    :  IF ((DI[26] OR DI[27]) AND F[324]),JMP LBL[53] ;
    :  IF ((!F[324] OR (TIMER[8]>=0)) AND ((F[523] AND !F[524] AND DI[2161]) OR (!F[523] AND F[524] AND !DI[2162])) AND DI[2167] AND F[576]),JMP LBL[54] ;
    :  IF ((!F[324] OR (TIMER[8]>=0)) AND ((F[523] AND !F[524] AND DI[2161]) OR (!F[523] AND F[524] AND !DI[2162])) AND !DI[2167] AND !F[576]),JMP LBL[54] ;
    :  R[42]=53    ;
    :   ;
    :  !**************************** ;
    :  !*        Schritt 54        * ;
    :  !*       MS1 Reinigung      * ;
    :  !* MS1 in Ruhest. schwenken * ;
    :  !**************************** ;
    :   ;
    :  LBL[54] ;
    :  R[41]=54    ;
    :  DO[2167]=(OFF) ;
    :  !Steuerluft EIN ;
    :  DO[2161]=(ON) ;
    :  !Schwenkeinheit 1 in Ruhestellung ;
    :  DO[2163]=(!DI[2163]) ;
    :  DO[2164]=(OFF) ;
    :  !FRG Bewegung EIN ;
    :  DO[2165]=(OFF) ;
    :  DO[2166]=(!DI[2163]) ;
    :  DO[18181]=(ON) ;
    :  WAIT (!DI[2164] AND DI[2163])    ;
    :  DO[18181]=(OFF) ;
    :  !RSK Fehlerausgabe Schwenkeinheit ;
    :  F[323]=((!DI[2163] AND (TIMER[8]>=0)) OR F[323]) ;
    :  !RSK Sammelstoerung ;
    :  F[329]=(F[323]) ;
    :  DO[2163]=(OFF) ;
    :  DO[2164]=(OFF) ;
    :  !FRG Bewegung AUS ;
    :  DO[2166]=(OFF) ;
    :  IF (F[323] AND (DI[26] OR DI[27])),JMP LBL[47] ;
    :  DO[18181]=(ON) ;
    :  WAIT (!F[323] AND DI[2165])    ;
    :  DO[18181]=(OFF) ;
    :  F[323]=(OFF) ;
    :  F[329]=(OFF) ;
    :  !FRG in Endlage halten ein ;
    :  DO[2165]=(ON) ;
    :  DO[18181]=(ON) ;
    :  WAIT   2.00(sec) ;
    :  WAIT (!DI[2165])    ;
    :  DO[18181]=(OFF) ;
    :  !Steuerluft AUS ;
    :  DO[2161]=(OFF) ;
    :  !FRG in Endlage halten AUS ;
    :  DO[2165]=(OFF) ;
    :  !MS1 Zaehler ruecksetzen ;
    :  R[21]=0    ;
    :  !MS1 FRG Reinigung ;
    :  F[603]=(OFF) ;
    :  !MS1 Reinigung FK ;
    :  F[605]=(ON) ;
    :  R[42]=54    ;
    :  JMP LBL[1] ;
    :   ;
    :  !************************** ;
    :  !*       Schritt 55       * ;
    :  !*      STAT EZ1/SP1      * ;
    :  !* 2.Setzhub nach Fraesen * ;
    :  !************************** ;
    :   ;
    :  LBL[55] ;
    :  R[41]=55    ;
    :  !RSK gestartet ;
    :  F[321]=(OFF) ;
    :  !EZ1/SK1 Prog. ;
    :  IF (F[78]),GO[1]=(61) ;
    :  IF (F[78]),GO[3]=(61) ;
    :  WAIT    .10(sec) ;
    :  !EZ1/SP1 schliessen ;
    :  DO[717]=(OFF) ;
    :  DO[718]=(ON) ;
    :  TIMER[9]=((-8)) ;
    :  !EZ1/SP1 Kraft erreicht ;
    :  WAIT ((DI[718] AND !DI[717]) OR (TIMER[9]>=0))    ;
    :  DO[18181]=((TIMER[9]>=0)) ;
    :  WAIT (DI[718] AND !DI[717])    ;
    :  DO[18181]=(OFF) ;
    :  WAIT   1.00(sec) ;
    :  !EZ1/SP1 oeffnen ;
    :  DO[718]=(OFF) ;
    :  DO[717]=(!DI[717]) ;
    :  TIMER[9]=((-8)) ;
    :  WAIT (DI[717] OR (TIMER[9]>=0))    ;
    :  DO[18181]=((TIMER[9]>=0)) ;
    :  WAIT (DI[717])    ;
    :  DO[18181]=(OFF) ;
    :  DO[717]=(OFF) ;
    :  R[42]=55    ;
    :  JMP LBL[16] ;
    :   ;
    :  !************************** ;
    :  !*       Schritt 56       * ;
    :  !*      STAT EZ2/SP2      * ;
    :  !* 2.Setzhub nach Fraesen * ;
    :  !************************** ;
    :   ;
    :  LBL[56] ;
    :  R[41]=56    ;
    :  !RSK gestartet ;
    :  F[321]=(OFF) ;
    :  !EZ2/SK2 Prog. ;
    :  IF (F[285] AND F[138]),GO[3]=(65) ;
    :  IF (!F[285] AND F[138]),GO[4]=(61) ;
    :  IF (!F[285] AND F[138]),GO[6]=(61) ;
    :  WAIT    .10(sec) ;
    :  !EZ2/SP2 schliessen ;
    :  DO[877]=(OFF) ;
    :  DO[878]=(ON) ;
    :  TIMER[9]=((-8)) ;
    :  !EZ2/SP2 Kraft erreicht ;
    :  WAIT ((DI[878] AND !DI[877]) OR (TIMER[9]>=0))    ;
    :  DO[18181]=((TIMER[9]>=0)) ;
    :  WAIT (DI[878] AND !DI[877])    ;
    :  DO[18181]=(OFF) ;
    :  WAIT   1.00(sec) ;
    :  !EZ2/SP2 oeffnen ;
    :  DO[878]=(OFF) ;
    :  DO[877]=(!DI[877]) ;
    :  TIMER[9]=((-8)) ;
    :  WAIT (DI[877] OR (TIMER[9]>=0))    ;
    :  DO[18181]=((TIMER[9]>=0)) ;
    :  WAIT (DI[877])    ;
    :  DO[18181]=(OFF) ;
    :  DO[877]=(OFF) ;
    :  R[42]=56    ;
    :  JMP LBL[25] ;
    :   ;
    :  !************************** ;
    :  !*       Schritt 57       * ;
    :  !*      STAT EZ3/SP3      * ;
    :  !* 2.Setzhub nach Fraesen * ;
    :  !************************** ;
    :   ;
    :  LBL[57] ;
    :  R[41]=57    ;
    :  !RSK gestartet ;
    :  F[321]=(OFF) ;
    :  !EZ1/SK1 Prog. ;
    :  IF (F[174]),GO[7]=(61) ;
    :  IF (F[174]),GO[9]=(61) ;
    :  WAIT    .10(sec) ;
    :  !EZ3/SP3 schliessen ;
    :  DO[1037]=(OFF) ;
    :  DO[1038]=(ON) ;
    :  TIMER[9]=((-8)) ;
    :  !EZ3/SP3 Kraft erreicht ;
    :  WAIT ((DI[1038] AND !DI[1037]) OR (TIMER[9]>=0))    ;
    :  DO[18181]=((TIMER[9]>=0)) ;
    :  WAIT (DI[1038] AND !DI[1037])    ;
    :  DO[18181]=(OFF) ;
    :  WAIT   1.00(sec) ;
    :  !EZ3/SP3 oeffnen ;
    :  DO[1038]=(OFF) ;
    :  DO[1037]=(!DI[1037]) ;
    :  TIMER[9]=((-8)) ;
    :  WAIT (DI[1037] OR (TIMER[9]>=0))    ;
    :  DO[18181]=((TIMER[9]>=0)) ;
    :  WAIT (DI[1037])    ;
    :  DO[18181]=(OFF) ;
    :  DO[1037]=(OFF) ;
    :  R[42]=57    ;
    :  JMP LBL[34] ;
    :   ;
    :  !*************************** ;
    :  !*************************** ;
    :  !* Fraesen Rob EZ1 SZ1-SZ4 * ;
    :  !*          an KF2         * ;
    :  !*************************** ;
    :  !*************************** ;
    :   ;
    :   ;
    :  !**************************** ;
    :  !*        Schritt 58        * ;
    :  !* Rob EZ1 SZ1-SZ4 Auswert. * ;
    :  !**************************** ;
    :   ;
    :  LBL[58] ;
    :  R[41]=58    ;
    :  !RSK gestartet ;
    :  F[321]=(OFF) ;
    :  GO[1]=(31) ;
    :  IF (F[64]),GO[3]=(31) ;
    :  IF (F[65]),GO[3]=(32) ;
    :  IF (F[66]),GO[3]=(33) ;
    :  IF (F[67]),GO[3]=(34) ;
    :  WAIT    .10(sec) ;
    :  DO[116]=(ON) ;
    :  DO[130]=(ON) ;
    :  DO[718]=(OFF) ;
    :  DO[717]=(!DI[717]) ;
    :  DO[18181]=(ON) ;
    :  WAIT (DI[717])    ;
    :  DO[18181]=(OFF) ;
    :  DO[717]=(OFF) ;
    :  !Anwahl Startfraesen ;
    :  IF (F[90] AND F[78] AND !F[79]),R[41]=59 ;
    :  !Anwahl Normalfraesen ;
    :  IF (F[90] AND !F[78] AND F[79]),R[41]=61 ;
    :  R[42]=58    ;
    :  JMP LBL[R[41]] ;
    :   ;
    :  !***************************** ;
    :  !*         Schritt 59        * ;
    :  !* Rob EZ1 SZ1-SZ4 SF Teil 1 * ;
    :  !***************************** ;
    :   ;
    :  LBL[59] ;
    :  R[41]=59    ;
    :  !RSK gestartet ;
    :  F[321]=(OFF) ;
    :  F[329]=(OFF) ;
    :  F[325]=(OFF) ;
    :  DO[718]=(OFF) ;
    :  DO[717]=(!DI[717]) ;
    :  DO[18181]=(ON) ;
    :  WAIT (DI[717])    ;
    :  DO[18181]=(OFF) ;
    :  DO[994]=(ON) ;
    :  DO[717]=(OFF) ;
    :  !Warte Fraeser laeuft ;
    :  TIMER[7]=((-3)) ;
    :  WAIT (!DI[994] OR (TIMER[7]>=0))    ;
    :  WAIT (DI[994] OR (TIMER[7]>=0))    ;
    :  F[322]=((TIMER[7]>=0)) ;
    :  DO[18181]=(ON) ;
    :  WAIT (!DI[994])    ;
    :  WAIT (DI[994])    ;
    :  DO[18181]=(OFF) ;
    :  F[322]=(OFF) ;
    :  !EZ1/SP1 schliessen ;
    :  DO[718]=(ON) ;
    :  TIMER[9]=((-4)) ;
    :  !EZ1/SP1 Kraft erreicht ;
    :  WAIT ((DI[718] AND !DI[772] AND !DI[780] AND !DI[774] AND !DI[775]) OR (TIMER[9]>=0))    ;
    :  DO[18181]=(ON) ;
    :  DO[718]=((TIMER[9]<0)) ;
    :  DO[994]=((TIMER[9]<0)) ;
    :  WAIT ((DI[718] AND !DI[772] AND !DI[780] AND !DI[774] AND !DI[775]) OR DI[26] OR DI[27])    ;
    :  F[325]=(DI[26] OR DI[27]) ;
    :  DO[18181]=(OFF) ;
    :  !EZ1/SP1 Fehler Kraftaufbau ;
    :  IF (F[325]),JMP LBL[5906] ;
    :  TIMER[9]=((-5)) ;
    :  LBL[5900] ;
    :  WAIT (!DI[994] OR F[325] OR (TIMER[9]>=0))    ;
    :  WAIT (DI[994] OR F[325] OR (TIMER[9]>=0))    ;
    :  R[1]=(R[1]+1) ;
    :  F[329]=((TIMER[9]>=0)) ;
    :  !Fraeszeit ueberschritten ;
    :  IF (F[329]),JMP LBL[5906] ;
    :  IF (F[64]),JMP LBL[5902] ;
    :  IF (F[65]),JMP LBL[5903] ;
    :  IF (F[66]),JMP LBL[5904] ;
    :  IF (F[67]),JMP LBL[5905] ;
    :  !Umdrehungen Vergl.SZ1 ;
    :  LBL[5902] ;
    :  !Umdrehungen Vergleichen ;
    :  IF (R[1]<R[2]),JMP LBL[5900] ;
    :  JMP LBL[5901] ;
    :  !Umdrehungen Vergl.SZ2 ;
    :  LBL[5903] ;
    :  !Umdrehungen Vergleichen ;
    :  IF (R[1]<R[8]),JMP LBL[5900] ;
    :  JMP LBL[5901] ;
    :  !Umdrehungen Vergl.SZ3 ;
    :  LBL[5904] ;
    :  !Umdrehungen Vergleichen ;
    :  IF (R[1]<R[11]),JMP LBL[5900] ;
    :  JMP LBL[5901] ;
    :  !Umdrehungen Vergl.SZ4 ;
    :  LBL[5905] ;
    :  !Umdrehungen Vergleichen ;
    :  IF (R[1]<R[14]),JMP LBL[5900] ;
    :  JMP LBL[5901] ;
    :  LBL[5901] ;
    :  IF (F[64]),F[94]=(ON) ;
    :  IF (F[65]),F[100]=(ON) ;
    :  IF (F[66]),F[106]=(ON) ;
    :  IF (F[67]),F[112]=(ON) ;
    :  LBL[5906] ;
    :  DO[994]=((TIMER[9]<0)) ;
    :  !Fraeser ausblasen EIN ;
    :  DO[995]=((TIMER[9]<0)) ;
    :  DO[718]=(OFF) ;
    :  !EZ1/SP1 oeffnen ;
    :  DO[717]=(!DI[717]) ;
    :  DO[18181]=(F[329]) ;
    :  WAIT (!F[329] OR DI[26] OR DI[27])    ;
    :  DO[18181]=(OFF) ;
    :  DO[18181]=(ON) ;
    :  WAIT (DI[717])    ;
    :  DO[18181]=(OFF) ;
    :  DO[717]=(OFF) ;
    :  !Umdrehungen ruecksetzen ;
    :  R[1]=0    ;
    :  R[42]=59    ;
    :  IF (F[329] OR F[325]),JMP LBL[59] ;
    :  JMP LBL[60] ;
    :   ;
    :  !***************************** ;
    :  !*         Schritt 60        * ;
    :  !* Rob EZ1 SZ1-SZ4 SF Teil 2 * ;
    :  !***************************** ;
    :   ;
    :  LBL[60] ;
    :  R[41]=60    ;
    :  !RSK gestartet ;
    :  F[321]=(OFF) ;
    :  F[329]=(OFF) ;
    :  F[325]=(OFF) ;
    :  DO[718]=(OFF) ;
    :  DO[717]=(!DI[717]) ;
    :  DO[18181]=(ON) ;
    :  WAIT (DI[717])    ;
    :  DO[18181]=(OFF) ;
    :  DO[994]=(ON) ;
    :  DO[717]=(OFF) ;
    :  !EZ1/SP1 schliessen ;
    :  DO[718]=(ON) ;
    :  !Fraeser ausblasen AUS ;
    :  DO[995]=(OFF) ;
    :  TIMER[9]=((-4)) ;
    :  !EZ1/SP1 Kraft erreicht ;
    :  WAIT ((DI[718] AND !DI[772] AND !DI[780] AND !DI[774] AND !DI[775]) OR (TIMER[9]>=0))    ;
    :  DO[18181]=(ON) ;
    :  DO[718]=((TIMER[9]<0)) ;
    :  DO[994]=((TIMER[9]<0)) ;
    :  WAIT ((DI[718] AND !DI[772] AND !DI[780] AND !DI[774] AND !DI[775]) OR DI[26] OR DI[27])    ;
    :  F[325]=(DI[26] OR DI[27]) ;
    :  DO[18181]=(OFF) ;
    :  !EZ1/SP1 Fehler Kraftaufbau ;
    :  IF (F[325]),JMP LBL[60] ;
    :  TIMER[9]=((-5)) ;
    :  LBL[6000] ;
    :  WAIT (!DI[994] OR F[325] OR (TIMER[9]>=0))    ;
    :  WAIT (DI[994] OR F[325] OR (TIMER[9]>=0))    ;
    :  R[1]=(R[1]+1) ;
    :  F[329]=((TIMER[9]>=0)) ;
    :  !Fraeszeit ueberschritten ;
    :  IF (F[329]),JMP LBL[6006] ;
    :  IF (F[64]),JMP LBL[6002] ;
    :  IF (F[65]),JMP LBL[6003] ;
    :  IF (F[66]),JMP LBL[6004] ;
    :  IF (F[67]),JMP LBL[6005] ;
    :  !Umdrehungen Vergl.SZ1 ;
    :  LBL[6002] ;
    :  !Umdrehungen Vergleichen ;
    :  IF (R[1]<R[3]),JMP LBL[6000] ;
    :  JMP LBL[6001] ;
    :  !Umdrehungen Vergl.SZ2 ;
    :  LBL[6003] ;
    :  !Umdrehungen Vergleichen ;
    :  IF (R[1]<R[9]),JMP LBL[6000] ;
    :  JMP LBL[6001] ;
    :  !Umdrehungen Vergl.SZ3 ;
    :  LBL[6004] ;
    :  !Umdrehungen Vergleichen ;
    :  IF (R[1]<R[12]),JMP LBL[6000] ;
    :  JMP LBL[6001] ;
    :  !Umdrehungen Vergl.SZ4 ;
    :  LBL[6005] ;
    :  !Umdrehungen Vergleichen ;
    :  IF (R[1]<R[15]),JMP LBL[6000] ;
    :  JMP LBL[6001] ;
    :  LBL[6001] ;
    :  IF (F[64]),F[96]=(ON) ;
    :  IF (F[65]),F[102]=(ON) ;
    :  IF (F[66]),F[108]=(ON) ;
    :  IF (F[67]),F[114]=(ON) ;
    :  LBL[6006] ;
    :  DO[994]=((TIMER[9]<0)) ;
    :  !Fraeser ausblasen EIN ;
    :  IF ((TIMER[9]<0)),DO[995]=PULSE,3.0sec ;
    :  DO[718]=(OFF) ;
    :  !EZ1/SP1 oeffnen ;
    :  DO[717]=(!DI[717]) ;
    :  DO[18181]=(F[329]) ;
    :  WAIT (!F[329] OR DI[26] OR DI[27])    ;
    :  DO[18181]=(OFF) ;
    :  DO[18181]=(ON) ;
    :  WAIT (DI[717])    ;
    :  DO[18181]=(OFF) ;
    :  DO[717]=(OFF) ;
    :  !Umdrehungen ruecksetzen ;
    :  R[1]=0    ;
    :  R[42]=60    ;
    :  IF (F[329] OR F[325]),JMP LBL[60] ;
    :  JMP LBL[62] ;
    :   ;
    :  !********************** ;
    :  !*     Schritt 61      * ;
    :  !* Rob EZ1 SZ1-SZ4 NF * ;
    :  !********************** ;
    :   ;
    :  LBL[61] ;
    :  R[41]=61    ;
    :  !RSK gestartet ;
    :  F[321]=(OFF) ;
    :  F[329]=(OFF) ;
    :  F[325]=(OFF) ;
    :  DO[718]=(OFF) ;
    :  DO[717]=(!DI[717]) ;
    :  DO[18181]=(ON) ;
    :  WAIT (DI[717])    ;
    :  DO[18181]=(OFF) ;
    :  DO[994]=(ON) ;
    :  DO[717]=(OFF) ;
    :  !Warte Fraeser laeuft ;
    :  TIMER[7]=((-3)) ;
    :  WAIT (!DI[994] OR (TIMER[7]>=0))    ;
    :  WAIT (DI[994] OR (TIMER[7]>=0))    ;
    :  F[322]=((TIMER[7]>=0)) ;
    :  DO[18181]=(ON) ;
    :  WAIT (!DI[994])    ;
    :  WAIT (DI[994])    ;
    :  DO[18181]=(OFF) ;
    :  F[322]=(OFF) ;
    :  !EZ1/SP1 schliessen ;
    :  DO[718]=(ON) ;
    :  TIMER[9]=((-4)) ;
    :  !EZ1/SP1 Kraft erreicht ;
    :  WAIT ((DI[718] AND !DI[772] AND !DI[780] AND !DI[774] AND !DI[775]) OR (TIMER[9]>=0))    ;
    :  DO[18181]=(ON) ;
    :  DO[718]=((TIMER[9]<0)) ;
    :  DO[994]=((TIMER[9]<0)) ;
    :  WAIT ((DI[718] AND !DI[772] AND !DI[780] AND !DI[774] AND !DI[775]) OR DI[26] OR DI[27])    ;
    :  F[325]=(DI[26] OR DI[27]) ;
    :  DO[18181]=(OFF) ;
    :  !EZ1/SP1 Fehler Kraftaufbau ;
    :  IF (F[325]),JMP LBL[61] ;
    :  TIMER[9]=((-5)) ;
    :  LBL[6100] ;
    :  WAIT (!DI[994] OR F[325] OR (TIMER[9]>=0))    ;
    :  WAIT (DI[994] OR F[325] OR (TIMER[9]>=0))    ;
    :  R[1]=(R[1]+1) ;
    :  F[329]=((TIMER[9]>=0)) ;
    :  !Fraeszeit ueberschritten ;
    :  IF (F[329]),JMP LBL[6106] ;
    :  IF (F[64]),JMP LBL[6102] ;
    :  IF (F[65]),JMP LBL[6103] ;
    :  IF (F[66]),JMP LBL[6104] ;
    :  IF (F[67]),JMP LBL[6105] ;
    :  !Umdrehungen Vergl.SZ1 ;
    :  LBL[6102] ;
    :  !Umdrehungen Vergleichen ;
    :  IF (R[1]<R[4]),JMP LBL[6100] ;
    :  JMP LBL[6101] ;
    :  !Umdrehungen Vergl.SZ2 ;
    :  LBL[6103] ;
    :  !Umdrehungen Vergleichen ;
    :  IF (R[1]<R[10]),JMP LBL[6100] ;
    :  !Umdrehungen Vergl.SZ3 ;
    :  LBL[6104] ;
    :  !Umdrehungen Vergleichen ;
    :  IF (R[1]<R[13]),JMP LBL[6100] ;
    :  JMP LBL[6101] ;
    :  !Umdrehungen Vergl.SZ4 ;
    :  LBL[6105] ;
    :  !Umdrehungen Vergleichen ;
    :  IF (R[1]<R[16]),JMP LBL[6100] ;
    :  LBL[6101] ;
    :  !EZ1/SP1 2 Huebe bei NF ;
    :  IF (!F[130]),JMP LBL[6106] ;
    :  IF (F[98]),F[96]=(ON) ;
    :  IF (F[104]),F[96]=(ON) ;
    :  IF (F[110]),F[96]=(ON) ;
    :  IF (F[116]),F[96]=(ON) ;
    :  IF (F[64]),F[98]=(ON) ;
    :  IF (F[65]),F[104]=(ON) ;
    :  IF (F[66]),F[110]=(ON) ;
    :  IF (F[67]),F[116]=(ON) ;
    :  LBL[6106] ;
    :  DO[994]=((TIMER[9]<0)) ;
    :  !Fraeser ausblasen EIN ;
    :  IF ((TIMER[9]<0)),DO[995]=PULSE,3.0sec ;
    :  DO[718]=(OFF) ;
    :  !EZ1/SP1 oeffnen ;
    :  DO[717]=(!DI[717]) ;
    :  DO[18181]=(F[329]) ;
    :  WAIT (!F[329] OR DI[26] OR DI[27])    ;
    :  DO[18181]=(OFF) ;
    :  DO[18181]=(ON) ;
    :  WAIT (DI[717])    ;
    :  DO[18181]=(OFF) ;
    :  DO[717]=(OFF) ;
    :  !Umdrehungen ruecksetzen ;
    :  R[1]=0    ;
    :  R[42]=61    ;
    :  IF (F[329] OR (!F[96] AND F[130])),JMP LBL[61] ;
    :  IF (F[64]),F[98]=(ON) ;
    :  IF (F[65]),F[104]=(ON) ;
    :  IF (F[66]),F[110]=(ON) ;
    :  IF (F[67]),F[116]=(ON) ;
    :  JMP LBL[62] ;
    :   ;
    :  !******************************* ;
    :  !*         Schritt 62          * ;
    :  !* Rob EZ1 SZ1-SZ4 i.O./n.i.O. * ;
    :  !******************************* ;
    :   ;
    :  LBL[62] ;
    :  R[41]=62    ;
    :  !Fraesueberwachung starten ;
    :  IF (F[64]),JMP LBL[6201] ;
    :  IF (F[65]),JMP LBL[6202] ;
    :  IF (F[66]),JMP LBL[6203] ;
    :  IF (F[67]),JMP LBL[6204] ;
    :  LBL[6201] ;
    :  TIMER[7]=((-3)) ;
    :  WAIT (F[64] AND ((F[79] AND F[98]) OR (F[78] AND F[94] AND F[96])) OR (TIMER[7]>=0))    ;
    :  F[329]=((TIMER[7]>=0)) ;
    :  DO[18181]=(ON) ;
    :  WAIT (F[64] AND ((F[79] AND F[98]) OR (F[78] AND F[94] AND F[96])))    ;
    :  DO[18181]=(OFF) ;
    :  JMP LBL[6200] ;
    :  LBL[6202] ;
    :  TIMER[7]=((-3)) ;
    :  WAIT (F[65] AND ((F[79] AND F[104]) OR (F[78] AND F[100] AND F[102])) OR (TIMER[7]>=0))    ;
    :  F[329]=((TIMER[7]>=0)) ;
    :  DO[18181]=(ON) ;
    :  WAIT (F[65] AND ((F[79] AND F[104]) OR (F[78] AND F[100] AND F[102])))    ;
    :  DO[18181]=(OFF) ;
    :  JMP LBL[6200] ;
    :  LBL[6203] ;
    :  TIMER[7]=((-3)) ;
    :  WAIT (F[66] AND ((F[79] AND F[110]) OR (F[78] AND F[106] AND F[108])) OR (TIMER[7]>=0))    ;
    :  F[329]=((TIMER[7]>=0)) ;
    :  DO[18181]=(ON) ;
    :  WAIT (F[66] AND ((F[79] AND F[110]) OR (F[78] AND F[106] AND F[108])))    ;
    :  DO[18181]=(OFF) ;
    :  JMP LBL[6200] ;
    :  LBL[6204] ;
    :  TIMER[7]=((-3)) ;
    :  WAIT (F[67] AND ((F[79] AND F[116]) OR (F[78] AND F[112] AND F[114])) OR (TIMER[7]>=0))    ;
    :  F[329]=((TIMER[7]>=0)) ;
    :  DO[18181]=(ON) ;
    :  WAIT (F[67] AND ((F[79] AND F[116]) OR (F[78] AND F[112] AND F[114])))    ;
    :  DO[18181]=(OFF) ;
    :  JMP LBL[6200] ;
    :  LBL[6200] ;
    :  R[41]=63    ;
    :  !KF1 U-Merker ruecksetzen ;
    :  F[94]=(OFF) ;
    :  F[96]=(OFF) ;
    :  F[98]=(OFF) ;
    :  F[100]=(OFF) ;
    :  F[102]=(OFF) ;
    :  F[104]=(OFF) ;
    :  F[106]=(OFF) ;
    :  F[108]=(OFF) ;
    :  F[110]=(OFF) ;
    :  F[112]=(OFF) ;
    :  F[114]=(OFF) ;
    :  F[116]=(OFF) ;
    :  R[42]=62    ;
    :  JMP LBL[R[41]] ;
    :   ;
    :  !***************************** ;
    :  !*        Schritt 63         * ;
    :  !* Rob EZ1 SZ1-SZ4 Quitt SK1 * ;
    :  !***************************** ;
    :   ;
    :  LBL[63] ;
    :  R[41]=63    ;
    :  !RSK gestartet ;
    :  F[321]=(OFF) ;
    :  IF (F[64]),GO[3]=1 ;
    :  IF (F[65]),GO[3]=2 ;
    :  IF (F[66]),GO[3]=3 ;
    :  IF (F[67]),GO[3]=4 ;
    :  WAIT    .10(sec) ;
    :  DO[786]=(ON) ;
    :  DO[116]=(OFF) ;
    :  DO[130]=(OFF) ;
    :  DO[18181]=(ON) ;
    :  WAIT (!DI[786] AND DI[787] AND !DI[788])    ;
    :  !FK Fraesen ;
    :  F[91]=(!F[329]) ;
    :  DO[18181]=(OFF) ;
    :  DO[786]=(OFF) ;
    :  R[42]=63    ;
    :  JMP LBL[1] ;
    :   ;
    :  !*************************** ;
    :  !*************************** ;
    :  !* Fraesen Rob EZ1 SZ1-SZ4 * ;
    :  !*          an KF3         * ;
    :  !*************************** ;
    :  !*************************** ;
    :   ;
    :   ;
    :  !**************************** ;
    :  !*        Schritt 64        * ;
    :  !* Rob EZ1 SZ1-SZ4 Auswert. * ;
    :  !**************************** ;
    :   ;
    :  LBL[64] ;
    :  R[41]=64    ;
    :  !RSK gestartet ;
    :  F[321]=(OFF) ;
    :  GO[1]=(31) ;
    :  IF (F[64]),GO[3]=(31) ;
    :  IF (F[65]),GO[3]=(32) ;
    :  IF (F[66]),GO[3]=(33) ;
    :  IF (F[67]),GO[3]=(34) ;
    :  WAIT    .10(sec) ;
    :  DO[116]=(ON) ;
    :  DO[130]=(ON) ;
    :  DO[718]=(OFF) ;
    :  DO[717]=(!DI[717]) ;
    :  DO[18181]=(ON) ;
    :  WAIT (DI[717])    ;
    :  DO[18181]=(OFF) ;
    :  DO[717]=(OFF) ;
    :  !Anwahl Startfraesen ;
    :  IF (F[90] AND F[78] AND !F[79]),R[41]=65 ;
    :  !Anwahl Normalfraesen ;
    :  IF (F[90] AND !F[78] AND F[79]),R[41]=67 ;
    :  R[42]=64    ;
    :  JMP LBL[R[41]] ;
    :   ;
    :  !***************************** ;
    :  !*         Schritt 65        * ;
    :  !* Rob EZ1 SZ1-SZ4 SF Teil 1 * ;
    :  !***************************** ;
    :   ;
    :  LBL[65] ;
    :  R[41]=65    ;
    :  !RSK gestartet ;
    :  F[321]=(OFF) ;
    :  F[329]=(OFF) ;
    :  F[325]=(OFF) ;
    :  DO[718]=(OFF) ;
    :  DO[717]=(!DI[717]) ;
    :  DO[18181]=(ON) ;
    :  WAIT (DI[717])    ;
    :  DO[18181]=(OFF) ;
    :  DO[1154]=(ON) ;
    :  DO[717]=(OFF) ;
    :  !Warte Fraeser laeuft ;
    :  TIMER[7]=((-3)) ;
    :  WAIT (!DI[1154] OR (TIMER[7]>=0))    ;
    :  WAIT (DI[1154] OR (TIMER[7]>=0))    ;
    :  F[322]=((TIMER[7]>=0)) ;
    :  DO[18181]=(ON) ;
    :  WAIT (!DI[1154])    ;
    :  WAIT (DI[1154])    ;
    :  DO[18181]=(OFF) ;
    :  F[322]=(OFF) ;
    :  !EZ1/SP1 schliessen ;
    :  DO[718]=(ON) ;
    :  TIMER[9]=((-4)) ;
    :  !EZ1/SP1 Kraft erreicht ;
    :  WAIT ((DI[718] AND !DI[772] AND !DI[780] AND !DI[774] AND !DI[775]) OR (TIMER[9]>=0))    ;
    :  DO[18181]=(ON) ;
    :  DO[718]=((TIMER[9]<0)) ;
    :  DO[1154]=((TIMER[9]<0)) ;
    :  WAIT ((DI[718] AND !DI[772] AND !DI[780] AND !DI[774] AND !DI[775]) OR DI[26] OR DI[27])    ;
    :  F[325]=(DI[26] OR DI[27]) ;
    :  DO[18181]=(OFF) ;
    :  !EZ1/SP1 Fehler Kraftaufbau ;
    :  IF (F[325]),JMP LBL[6506] ;
    :  TIMER[9]=((-5)) ;
    :  LBL[6500] ;
    :  WAIT (!DI[1154] OR F[325] OR (TIMER[9]>=0))    ;
    :  WAIT (DI[1154] OR F[325] OR (TIMER[9]>=0))    ;
    :  R[1]=(R[1]+1) ;
    :  F[329]=((TIMER[9]>=0)) ;
    :  !Fraeszeit ueberschritten ;
    :  IF (F[329]),JMP LBL[6506] ;
    :  IF (F[64]),JMP LBL[6502] ;
    :  IF (F[65]),JMP LBL[6503] ;
    :  IF (F[66]),JMP LBL[6504] ;
    :  IF (F[67]),JMP LBL[6505] ;
    :  !Umdrehungen Vergl.SZ1 ;
    :  LBL[6502] ;
    :  !Umdrehungen Vergleichen ;
    :  IF (R[1]<R[2]),JMP LBL[6500] ;
    :  JMP LBL[6501] ;
    :  !Umdrehungen Vergl.SZ2 ;
    :  LBL[6503] ;
    :  !Umdrehungen Vergleichen ;
    :  IF (R[1]<R[8]),JMP LBL[6500] ;
    :  JMP LBL[6501] ;
    :  !Umdrehungen Vergl.SZ3 ;
    :  LBL[6504] ;
    :  !Umdrehungen Vergleichen ;
    :  IF (R[1]<R[11]),JMP LBL[6500] ;
    :  JMP LBL[6501] ;
    :  !Umdrehungen Vergl.SZ4 ;
    :  LBL[6505] ;
    :  !Umdrehungen Vergleichen ;
    :  IF (R[1]<R[14]),JMP LBL[6500] ;
    :  JMP LBL[6501] ;
    :  LBL[6501] ;
    :  IF (F[64]),F[94]=(ON) ;
    :  IF (F[65]),F[100]=(ON) ;
    :  IF (F[66]),F[106]=(ON) ;
    :  IF (F[67]),F[112]=(ON) ;
    :  LBL[6506] ;
    :  DO[1154]=((TIMER[9]<0)) ;
    :  !Fraeser ausblasen EIN ;
    :  DO[1155]=((TIMER[9]<0)) ;
    :  DO[718]=(OFF) ;
    :  !EZ1/SP1 oeffnen ;
    :  DO[717]=(!DI[717]) ;
    :  DO[18181]=(F[329]) ;
    :  WAIT (!F[329] OR DI[26] OR DI[27])    ;
    :  DO[18181]=(OFF) ;
    :  DO[18181]=(ON) ;
    :  WAIT (DI[717])    ;
    :  DO[18181]=(OFF) ;
    :  DO[717]=(OFF) ;
    :  !Umdrehungen ruecksetzen ;
    :  R[1]=0    ;
    :  R[42]=65    ;
    :  IF (F[329] OR F[325]),JMP LBL[65] ;
    :  JMP LBL[66] ;
    :   ;
    :  !***************************** ;
    :  !*         Schritt 66        * ;
    :  !* Rob EZ1 SZ1-SZ4 SF Teil 2 * ;
    :  !***************************** ;
    :   ;
    :  LBL[66] ;
    :  R[41]=66    ;
    :  !RSK gestartet ;
    :  F[321]=(OFF) ;
    :  F[329]=(OFF) ;
    :  F[325]=(OFF) ;
    :  DO[718]=(OFF) ;
    :  DO[717]=(!DI[717]) ;
    :  DO[18181]=(ON) ;
    :  WAIT (DI[717])    ;
    :  DO[18181]=(OFF) ;
    :  DO[1154]=(ON) ;
    :  DO[717]=(OFF) ;
    :  !EZ1/SP1 schliessen ;
    :  DO[718]=(ON) ;
    :  !Fraeser ausblasen AUS ;
    :  DO[1155]=(OFF) ;
    :  TIMER[9]=((-4)) ;
    :  !EZ1/SP1 Kraft erreicht ;
    :  WAIT ((DI[718] AND !DI[772] AND !DI[780] AND !DI[774] AND !DI[775]) OR (TIMER[9]>=0))    ;
    :  DO[18181]=(ON) ;
    :  DO[718]=((TIMER[9]<0)) ;
    :  DO[1154]=((TIMER[9]<0)) ;
    :  WAIT ((DI[718] AND !DI[772] AND !DI[780] AND !DI[774] AND !DI[775]) OR DI[26] OR DI[27])    ;
    :  F[325]=(DI[26] OR DI[27]) ;
    :  DO[18181]=(OFF) ;
    :  !EZ1/SP1 Fehler Kraftaufbau ;
    :  IF (F[325]),JMP LBL[66] ;
    :  TIMER[9]=((-5)) ;
    :  LBL[6600] ;
    :  WAIT (!DI[1154] OR F[325] OR (TIMER[9]>=0))    ;
    :  WAIT (DI[1154] OR F[325] OR (TIMER[9]>=0))    ;
    :  R[1]=(R[1]+1) ;
    :  F[329]=((TIMER[9]>=0)) ;
    :  !Fraeszeit ueberschritten ;
    :  IF (F[329]),JMP LBL[6606] ;
    :  IF (F[64]),JMP LBL[6602] ;
    :  IF (F[65]),JMP LBL[6603] ;
    :  IF (F[66]),JMP LBL[6604] ;
    :  IF (F[67]),JMP LBL[6605] ;
    :  !Umdrehungen Vergl.SZ1 ;
    :  LBL[6602] ;
    :  !Umdrehungen Vergleichen ;
    :  IF (R[1]<R[3]),JMP LBL[6600] ;
    :  JMP LBL[6601] ;
    :  !Umdrehungen Vergl.SZ2 ;
    :  LBL[6603] ;
    :  !Umdrehungen Vergleichen ;
    :  IF (R[1]<R[9]),JMP LBL[6600] ;
    :  JMP LBL[6601] ;
    :  !Umdrehungen Vergl.SZ3 ;
    :  LBL[6604] ;
    :  !Umdrehungen Vergleichen ;
    :  IF (R[1]<R[12]),JMP LBL[6600] ;
    :  JMP LBL[6601] ;
    :  !Umdrehungen Vergl.SZ4 ;
    :  LBL[6605] ;
    :  !Umdrehungen Vergleichen ;
    :  IF (R[1]<R[15]),JMP LBL[6600] ;
    :  JMP LBL[6601] ;
    :  LBL[6601] ;
    :  IF (F[64]),F[96]=(ON) ;
    :  IF (F[65]),F[102]=(ON) ;
    :  IF (F[66]),F[108]=(ON) ;
    :  IF (F[67]),F[114]=(ON) ;
    :  LBL[6606] ;
    :  DO[1154]=((TIMER[9]<0)) ;
    :  !Fraeser ausblasen EIN ;
    :  IF ((TIMER[9]<0)),DO[1155]=PULSE,3.0sec ;
    :  DO[718]=(OFF) ;
    :  !EZ1/SP1 oeffnen ;
    :  DO[717]=(!DI[717]) ;
    :  DO[18181]=(F[329]) ;
    :  WAIT (!F[329] OR DI[26] OR DI[27])    ;
    :  DO[18181]=(OFF) ;
    :  DO[18181]=(ON) ;
    :  WAIT (DI[717])    ;
    :  DO[18181]=(OFF) ;
    :  DO[717]=(OFF) ;
    :  !Umdrehungen ruecksetzen ;
    :  R[1]=0    ;
    :  R[42]=66    ;
    :  IF (F[329] OR F[325]),JMP LBL[66] ;
    :  JMP LBL[68] ;
    :   ;
    :  !********************** ;
    :  !*     Schritt 67     * ;
    :  !* Rob EZ1 SZ1-SZ4 NF * ;
    :  !********************** ;
    :   ;
    :  LBL[67] ;
    :  R[41]=67    ;
    :  !RSK gestartet ;
    :  F[321]=(OFF) ;
    :  F[329]=(OFF) ;
    :  F[325]=(OFF) ;
    :  DO[718]=(OFF) ;
    :  DO[717]=(!DI[717]) ;
    :  DO[18181]=(ON) ;
    :  WAIT (DI[717])    ;
    :  DO[18181]=(OFF) ;
    :  DO[1154]=(ON) ;
    :  DO[717]=(OFF) ;
    :  !Warte Fraeser laeuft ;
    :  TIMER[7]=((-3)) ;
    :  WAIT (!DI[1154] OR (TIMER[7]>=0))    ;
    :  WAIT (DI[1154] OR (TIMER[7]>=0))    ;
    :  F[322]=((TIMER[7]>=0)) ;
    :  DO[18181]=(ON) ;
    :  WAIT (!DI[1154])    ;
    :  WAIT (DI[1154])    ;
    :  DO[18181]=(OFF) ;
    :  F[322]=(OFF) ;
    :  !EZ1/SP1 schliessen ;
    :  DO[718]=(ON) ;
    :  TIMER[9]=((-4)) ;
    :  !EZ1/SP1 Kraft erreicht ;
    :  WAIT ((DI[718] AND !DI[772] AND !DI[780] AND !DI[774] AND !DI[775]) OR (TIMER[9]>=0))    ;
    :  DO[18181]=(ON) ;
    :  DO[718]=((TIMER[9]<0)) ;
    :  DO[1154]=((TIMER[9]<0)) ;
    :  WAIT ((DI[718] AND !DI[772] AND !DI[780] AND !DI[774] AND !DI[775]) OR DI[26] OR DI[27])    ;
    :  F[325]=(DI[26] OR DI[27]) ;
    :  DO[18181]=(OFF) ;
    :  !EZ1/SP1 Fehler Kraftaufbau ;
    :  IF (F[325]),JMP LBL[67] ;
    :  TIMER[9]=((-5)) ;
    :  LBL[6700] ;
    :  WAIT (!DI[1154] OR F[325] OR (TIMER[9]>=0))    ;
    :  WAIT (DI[1154] OR F[325] OR (TIMER[9]>=0))    ;
    :  R[1]=(R[1]+1) ;
    :  F[329]=((TIMER[9]>=0)) ;
    :  !Fraeszeit ueberschritten ;
    :  IF (F[329]),JMP LBL[6706] ;
    :  IF (F[64]),JMP LBL[6702] ;
    :  IF (F[65]),JMP LBL[6703] ;
    :  IF (F[66]),JMP LBL[6704] ;
    :  IF (F[67]),JMP LBL[6705] ;
    :  !Umdrehungen Vergl.SZ1 ;
    :  LBL[6702] ;
    :  !Umdrehungen Vergleichen ;
    :  IF (R[1]<R[4]),JMP LBL[6700] ;
    :  JMP LBL[6701] ;
    :  !Umdrehungen Vergl.SZ2 ;
    :  LBL[6703] ;
    :  !Umdrehungen Vergleichen ;
    :  IF (R[1]<R[10]),JMP LBL[6700] ;
    :  !Umdrehungen Vergl.SZ3 ;
    :  LBL[6704] ;
    :  !Umdrehungen Vergleichen ;
    :  IF (R[1]<R[13]),JMP LBL[6700] ;
    :  JMP LBL[6701] ;
    :  !Umdrehungen Vergl.SZ4 ;
    :  LBL[6705] ;
    :  !Umdrehungen Vergleichen ;
    :  IF (R[1]<R[16]),JMP LBL[6700] ;
    :  LBL[6701] ;
    :  !EZ1/SP1 2 Huebe bei NF ;
    :  IF (!F[130]),JMP LBL[6706] ;
    :  IF (F[98]),F[96]=(ON) ;
    :  IF (F[104]),F[96]=(ON) ;
    :  IF (F[110]),F[96]=(ON) ;
    :  IF (F[116]),F[96]=(ON) ;
    :  IF (F[64]),F[98]=(ON) ;
    :  IF (F[65]),F[104]=(ON) ;
    :  IF (F[66]),F[110]=(ON) ;
    :  IF (F[67]),F[116]=(ON) ;
    :  LBL[6706] ;
    :  DO[1154]=((TIMER[9]<0)) ;
    :  !Fraeser ausblasen EIN ;
    :  IF ((TIMER[9]<0)),DO[1155]=PULSE,3.0sec ;
    :  DO[718]=(OFF) ;
    :  !EZ1/SP1 oeffnen ;
    :  DO[717]=(!DI[717]) ;
    :  DO[18181]=(F[329]) ;
    :  WAIT (!F[329] OR DI[26] OR DI[27])    ;
    :  DO[18181]=(OFF) ;
    :  DO[18181]=(ON) ;
    :  WAIT (DI[717])    ;
    :  DO[18181]=(OFF) ;
    :  DO[717]=(OFF) ;
    :  !Umdrehungen ruecksetzen ;
    :  R[1]=0    ;
    :  R[42]=67    ;
    :  IF (F[329] OR (!F[96] AND F[130])),JMP LBL[67] ;
    :  IF (F[64]),F[98]=(ON) ;
    :  IF (F[65]),F[104]=(ON) ;
    :  IF (F[66]),F[110]=(ON) ;
    :  IF (F[67]),F[116]=(ON) ;
    :  JMP LBL[68] ;
    :   ;
    :  !******************************* ;
    :  !*         Schritt 68           * ;
    :  !* Rob EZ1 SZ1-SZ4 i.O./n.i.O. * ;
    :  !******************************* ;
    :   ;
    :  LBL[68] ;
    :  R[41]=68    ;
    :  !Fraesueberwachung starten ;
    :  IF (F[64]),JMP LBL[6801] ;
    :  IF (F[65]),JMP LBL[6802] ;
    :  IF (F[66]),JMP LBL[6803] ;
    :  IF (F[67]),JMP LBL[6804] ;
    :  LBL[6801] ;
    :  TIMER[7]=((-3)) ;
    :  WAIT (F[64] AND ((F[79] AND F[98]) OR (F[78] AND F[94] AND F[96])) OR (TIMER[7]>=0))    ;
    :  F[329]=((TIMER[7]>=0)) ;
    :  DO[18181]=(ON) ;
    :  WAIT (F[64] AND ((F[79] AND F[98]) OR (F[78] AND F[94] AND F[96])))    ;
    :  DO[18181]=(OFF) ;
    :  JMP LBL[6800] ;
    :  LBL[6802] ;
    :  TIMER[7]=((-3)) ;
    :  WAIT (F[65] AND ((F[79] AND F[104]) OR (F[78] AND F[100] AND F[102])) OR (TIMER[7]>=0))    ;
    :  F[329]=((TIMER[7]>=0)) ;
    :  DO[18181]=(ON) ;
    :  WAIT (F[65] AND ((F[79] AND F[104]) OR (F[78] AND F[100] AND F[102])))    ;
    :  DO[18181]=(OFF) ;
    :  JMP LBL[6800] ;
    :  LBL[6803] ;
    :  TIMER[7]=((-3)) ;
    :  WAIT (F[66] AND ((F[79] AND F[110]) OR (F[78] AND F[106] AND F[108])) OR (TIMER[7]>=0))    ;
    :  F[329]=((TIMER[7]>=0)) ;
    :  DO[18181]=(ON) ;
    :  WAIT (F[66] AND ((F[79] AND F[110]) OR (F[78] AND F[106] AND F[108])))    ;
    :  DO[18181]=(OFF) ;
    :  JMP LBL[6800] ;
    :  LBL[6804] ;
    :  TIMER[7]=((-3)) ;
    :  WAIT (F[67] AND ((F[79] AND F[116]) OR (F[78] AND F[112] AND F[114])) OR (TIMER[7]>=0))    ;
    :  F[329]=((TIMER[7]>=0)) ;
    :  DO[18181]=(ON) ;
    :  WAIT (F[67] AND ((F[79] AND F[116]) OR (F[78] AND F[112] AND F[114])))    ;
    :  DO[18181]=(OFF) ;
    :  JMP LBL[6800] ;
    :  LBL[6800] ;
    :  R[41]=69    ;
    :  !KF1 U-Merker ruecksetzen ;
    :  F[94]=(OFF) ;
    :  F[96]=(OFF) ;
    :  F[98]=(OFF) ;
    :  F[100]=(OFF) ;
    :  F[102]=(OFF) ;
    :  F[104]=(OFF) ;
    :  F[106]=(OFF) ;
    :  F[108]=(OFF) ;
    :  F[110]=(OFF) ;
    :  F[112]=(OFF) ;
    :  F[114]=(OFF) ;
    :  F[116]=(OFF) ;
    :  R[42]=68    ;
    :  JMP LBL[R[41]] ;
    :   ;
    :  !***************************** ;
    :  !*        Schritt 69         * ;
    :  !* Rob EZ1 SZ1-SZ4 Quitt SK1 * ;
    :  !***************************** ;
    :   ;
    :  LBL[69] ;
    :  R[41]=69    ;
    :  !RSK gestartet ;
    :  F[321]=(OFF) ;
    :  IF (F[64]),GO[3]=1 ;
    :  IF (F[65]),GO[3]=2 ;
    :  IF (F[66]),GO[3]=3 ;
    :  IF (F[67]),GO[3]=4 ;
    :  WAIT    .10(sec) ;
    :  DO[786]=(ON) ;
    :  DO[116]=(OFF) ;
    :  DO[130]=(OFF) ;
    :  DO[18181]=(ON) ;
    :  WAIT (!DI[786] AND DI[787] AND !DI[788])    ;
    :  !FK Fraesen ;
    :  F[91]=(!F[329]) ;
    :  DO[18181]=(OFF) ;
    :  DO[786]=(OFF) ;
    :  R[42]=69    ;
    :  JMP LBL[1] ;
    :   ;
    :  !********************** ;
    :  !*     Schritt 70     * ;
    :  !* ROB STP1 SZ1 Start * ;
    :  !********************** ;
    :   ;
    :  LBL[70] ;
    :  R[41]=70    ;
    :  !RSK gestartet ;
    :  F[321]=(OFF) ;
    :  F[122]=(OFF) ;
    :  F[322]=(OFF) ;
    :  F[323]=(OFF) ;
    :  F[324]=(OFF) ;
    :  F[325]=(OFF) ;
    :  F[329]=(OFF) ;
    :  !Rob. STP1 SZ1 beim Fraesen ;
    :  DO[116]=(ON) ;
    :  DO[130]=(ON) ;
    :  !Anwahl Startfraesen ;
    :  IF (F[90] AND F[78] AND !F[79]),R[41]=71 ;
    :  !Anwahl Normalfraesen ;
    :  IF (F[90] AND !F[78] AND F[79]),R[41]=73 ;
    :  R[42]=70    ;
    :  JMP LBL[R[41]] ;
    :   ;
    :  !************************** ;
    :  !*      Schritt 71        * ;
    :  !* Rob STP1 SZ1 SF Teil 1 * ;
    :  !************************** ;
    :   ;
    :  LBL[71] ;
    :  R[41]=71    ;
    :  !RSK gestartet ;
    :  F[321]=(OFF) ;
    :  F[329]=(OFF) ;
    :  F[325]=(OFF) ;
    :  !KF1 einschalten ;
    :  DO[864]=(ON) ;
    :  !Warte Fraeser laeuft ;
    :  TIMER[7]=((-3)) ;
    :  WAIT (!DI[864] OR (TIMER[7]>=0))    ;
    :  WAIT (DI[864] OR (TIMER[7]>=0))    ;
    :  F[322]=((TIMER[7]>=0)) ;
    :  DO[18181]=(ON) ;
    :  WAIT (!DI[864])    ;
    :  WAIT (DI[864])    ;
    :  DO[18181]=(OFF) ;
    :  F[322]=(OFF) ;
    :  !KF1 hochfahren ;
    :  DO[863]=(ON) ;
    :  TIMER[8]=((-5)) ;
    :  WAIT (!DI[863] OR (TIMER[8]>=0))    ;
    :  F[324]=((TIMER[8]>=0)) ;
    :  DO[18181]=(ON) ;
    :  WAIT (!DI[863])    ;
    :  DO[18181]=(OFF) ;
    :  F[324]=(OFF) ;
    :  TIMER[9]=((-5)) ;
    :  LBL[7100] ;
    :  WAIT (!DI[864] OR (TIMER[9]>=0))    ;
    :  WAIT (DI[864] OR (TIMER[9]>=0))    ;
    :  R[1]=(R[1]+1) ;
    :  F[329]=((TIMER[9]>=0)) ;
    :  !Fraeszeit ueberschritten ;
    :  IF (F[329]),JMP LBL[7103] ;
    :  IF (F[64]),JMP LBL[7102] ;
    :  !Umdrehungen Vergl.SZ1 ;
    :  LBL[7102] ;
    :  !Umdrehungen Vergleichen ;
    :  IF (R[1]<R[2]),JMP LBL[7100] ;
    :  JMP LBL[7101] ;
    :  LBL[7101] ;
    :  IF (F[64]),F[94]=(ON) ;
    :  LBL[7103] ;
    :  DO[864]=(OFF) ;
    :  DO[18181]=(F[329]) ;
    :  WAIT (!F[329] OR DI[26] OR DI[27])    ;
    :  DO[18181]=(OFF) ;
    :  !KF1 runterfahren ;
    :  DO[863]=(OFF) ;
    :  TIMER[8]=((-5)) ;
    :  WAIT (DI[863] OR (TIMER[8]>=0))    ;
    :  F[324]=((TIMER[8]>=0)) ;
    :  DO[18181]=(ON) ;
    :  WAIT (DI[863])    ;
    :  DO[18181]=(OFF) ;
    :  F[324]=(OFF) ;
    :  !Umdrehungen ruecksetzen ;
    :  R[1]=0    ;
    :  R[42]=71    ;
    :  IF (F[329] OR F[325]),JMP LBL[71] ;
    :  JMP LBL[72] ;
    :   ;
    :  !************************** ;
    :  !*      Schritt 72        * ;
    :  !* Rob STP1 SZ1 SF Teil 2 * ;
    :  !************************** ;
    :   ;
    :  LBL[72] ;
    :  R[41]=72    ;
    :  !RSK gestartet ;
    :  F[321]=(OFF) ;
    :  F[329]=(OFF) ;
    :  F[325]=(OFF) ;
    :  !KF1 einschalten ;
    :  DO[864]=(ON) ;
    :  !Warte Fraeser laeuft ;
    :  TIMER[7]=((-3)) ;
    :  WAIT (!DI[864] OR (TIMER[7]>=0))    ;
    :  WAIT (DI[864] OR (TIMER[7]>=0))    ;
    :  F[322]=((TIMER[7]>=0)) ;
    :  DO[18181]=(ON) ;
    :  WAIT (!DI[864])    ;
    :  WAIT (DI[864])    ;
    :  DO[18181]=(OFF) ;
    :  F[322]=(OFF) ;
    :  !KF1 hochfahren ;
    :  DO[863]=(ON) ;
    :  TIMER[8]=((-5)) ;
    :  WAIT (!DI[863] OR (TIMER[8]>=0))    ;
    :  F[324]=((TIMER[8]>=0)) ;
    :  DO[18181]=(ON) ;
    :  WAIT (!DI[863])    ;
    :  DO[18181]=(OFF) ;
    :  F[324]=(OFF) ;
    :  TIMER[9]=((-5)) ;
    :  LBL[7200] ;
    :  WAIT (!DI[864] OR (TIMER[9]>=0))    ;
    :  WAIT (DI[864] OR (TIMER[9]>=0))    ;
    :  R[1]=(R[1]+1) ;
    :  F[329]=((TIMER[9]>=0)) ;
    :  !Fraeszeit ueberschritten ;
    :  IF (F[329]),JMP LBL[7203] ;
    :  IF (F[64]),JMP LBL[7202] ;
    :  !Umdrehungen Vergl.SZ1 ;
    :  LBL[7202] ;
    :  !Umdrehungen Vergleichen ;
    :  IF (R[1]<R[3]),JMP LBL[7200] ;
    :  JMP LBL[7201] ;
    :  LBL[7201] ;
    :  IF (F[64]),F[96]=(ON) ;
    :  LBL[7203] ;
    :  DO[864]=(OFF) ;
    :  DO[18181]=(F[329]) ;
    :  WAIT (!F[329] OR DI[26] OR DI[27])    ;
    :  DO[18181]=(OFF) ;
    :  !KF1 runterfahren ;
    :  DO[863]=(OFF) ;
    :  TIMER[8]=((-5)) ;
    :  WAIT (DI[863] OR (TIMER[8]>=0))    ;
    :  F[324]=((TIMER[8]>=0)) ;
    :  DO[18181]=(ON) ;
    :  WAIT (DI[863])    ;
    :  DO[18181]=(OFF) ;
    :  F[324]=(OFF) ;
    :  !Umdrehungen ruecksetzen ;
    :  R[1]=0    ;
    :  R[42]=73    ;
    :  IF (F[329] OR F[325]),JMP LBL[72] ;
    :  JMP LBL[73] ;
    :   ;
    :   ;
    :  !******************* ;
    :  !*   Schritt 73    * ;
    :  !* Rob STP1 SZ1 NF * ;
    :  !******************* ;
    :   ;
    :  LBL[73] ;
    :  R[41]=73    ;
    :  !RSK gestartet ;
    :  F[321]=(OFF) ;
    :  F[329]=(OFF) ;
    :  F[325]=(OFF) ;
    :  !KF1 einschalten ;
    :  DO[864]=(ON) ;
    :  !Warte Fraeser laeuft ;
    :  TIMER[7]=((-3)) ;
    :  WAIT (!DI[864] OR (TIMER[7]>=0))    ;
    :  WAIT (DI[864] OR (TIMER[7]>=0))    ;
    :  F[322]=((TIMER[7]>=0)) ;
    :  DO[18181]=(ON) ;
    :  WAIT (!DI[864])    ;
    :  WAIT (DI[864])    ;
    :  DO[18181]=(OFF) ;
    :  F[322]=(OFF) ;
    :  !KF1 hochfahren ;
    :  DO[863]=(ON) ;
    :  TIMER[8]=((-5)) ;
    :  WAIT (!DI[863] OR (TIMER[8]>=0))    ;
    :  F[324]=((TIMER[8]>=0)) ;
    :  DO[18181]=(ON) ;
    :  WAIT (!DI[863])    ;
    :  DO[18181]=(OFF) ;
    :  F[324]=(OFF) ;
    :  TIMER[9]=((-5)) ;
    :  LBL[7300] ;
    :  WAIT (!DI[864] OR (TIMER[9]>=0))    ;
    :  WAIT (DI[864] OR (TIMER[9]>=0))    ;
    :  R[1]=(R[1]+1) ;
    :  F[329]=((TIMER[9]>=0)) ;
    :  !Fraeszeit ueberschritten ;
    :  IF (F[329]),JMP LBL[7303] ;
    :  IF (F[64]),JMP LBL[7302] ;
    :  !Umdrehungen Vergl.SZ1 ;
    :  LBL[7302] ;
    :  !Umdrehungen Vergleichen ;
    :  IF (R[1]<R[4]),JMP LBL[7300] ;
    :  JMP LBL[7301] ;
    :  LBL[7301] ;
    :  IF (F[64]),F[98]=(ON) ;
    :  LBL[7303] ;
    :  DO[864]=(OFF) ;
    :  DO[18181]=(F[329]) ;
    :  WAIT (!F[329] OR DI[26] OR DI[27])    ;
    :  DO[18181]=(OFF) ;
    :  !KF1 runterfahren ;
    :  DO[863]=(OFF) ;
    :  TIMER[8]=((-5)) ;
    :  WAIT (DI[863] OR (TIMER[8]>=0))    ;
    :  F[324]=((TIMER[8]>=0)) ;
    :  DO[18181]=(ON) ;
    :  WAIT (DI[863])    ;
    :  DO[18181]=(OFF) ;
    :  F[324]=(OFF) ;
    :  !Umdrehungen ruecksetzen ;
    :  R[1]=0    ;
    :  R[42]=72    ;
    :  IF (F[329] OR F[325]),JMP LBL[73] ;
    :  JMP LBL[74] ;
    :   ;
    :  !*************************** ;
    :  !*       Schritt 74        * ;
    :  !* Rob STP SZ1 i.O./n.i.O. * ;
    :  !*************************** ;
    :   ;
    :  LBL[74] ;
    :  R[41]=74    ;
    :  !Fraesueberwachung starten ;
    :  TIMER[7]=((-3)) ;
    :  WAIT (F[64] AND ((F[79] AND F[98]) OR (F[78] AND F[94] AND F[96])) OR (TIMER[7]>=0))    ;
    :  F[329]=((TIMER[7]>=0)) ;
    :  DO[18181]=(ON) ;
    :  WAIT (F[64] AND ((F[79] AND F[98]) OR (F[78] AND F[94] AND F[96])))    ;
    :  DO[18181]=(OFF) ;
    :  R[41]=75    ;
    :  !KF1 U-Merker ruecksetzen ;
    :  F[94]=(OFF) ;
    :  F[96]=(OFF) ;
    :  F[98]=(OFF) ;
    :  R[42]=74    ;
    :  JMP LBL[R[41]] ;
    :   ;
    :  !***************************** ;
    :  !*        Schritt 75         * ;
    :  !*   Rob STP SZ1 Quitt SK1   * ;
    :  !***************************** ;
    :   ;
    :  LBL[75] ;
    :  R[41]=75    ;
    :  !RSK gestartet ;
    :  F[321]=(OFF) ;
    :  IF (F[64] AND !F[329]),GO[3]=1 ;
    :  WAIT    .10(sec) ;
    :  DO[786]=(!F[329] AND !F[322]) ;
    :  DO[18181]=(ON) ;
    :  WAIT ((!DI[786] AND DI[787] AND !DI[788] AND !F[329]) OR DI[26] OR DI[27])    ;
    :  !FK Fraesen ;
    :  F[91]=(!F[329]) ;
    :  DO[18181]=(OFF) ;
    :  DO[786]=(OFF) ;
    :  DO[116]=(OFF) ;
    :  DO[130]=(OFF) ;
    :  R[41]=1    ;
    :  IF (!F[329]),JMP LBL[7600] ;
    :  R[41]=70    ;
    :  LBL[7600] ;
    :  R[42]=75    ;
    :  JMP LBL[R[41]] ;
    :   ;
    :  !********************** ;
    :  !********************** ;
    :  !* Ende Makro_Schritt * ;
    :  !********************** ;
    :  !********************** ;
    :   ;
    :  !Loop fuer Makro_Schritt ;
    :  JMP LBL[1] ;
/POS
/END
